(* PLC project Unnamed, Unnamed Unnamed 1 *)
(* stored: creationDateTime 2024-11-22T14:37:36, modificationDateTime 2024-11-29T13:18:13 *)

PROGRAM Blink
  VAR
    blink_led : BOOL;
    TON0 : TON;
    TOF0 : TOF;
    LED_ON0 : LED_ON;
    LED_OFF0 : LED_OFF;
    LED_ON1 : LED_ON;
    LED_OFF1 : LED_OFF;
  END_VAR
  VAR  (* added by the conversion: wires and edge detectors of the diagram *)
    R_TRIG1 : R_TRIG;
    F_TRIG2 : F_TRIG;
  END_VAR

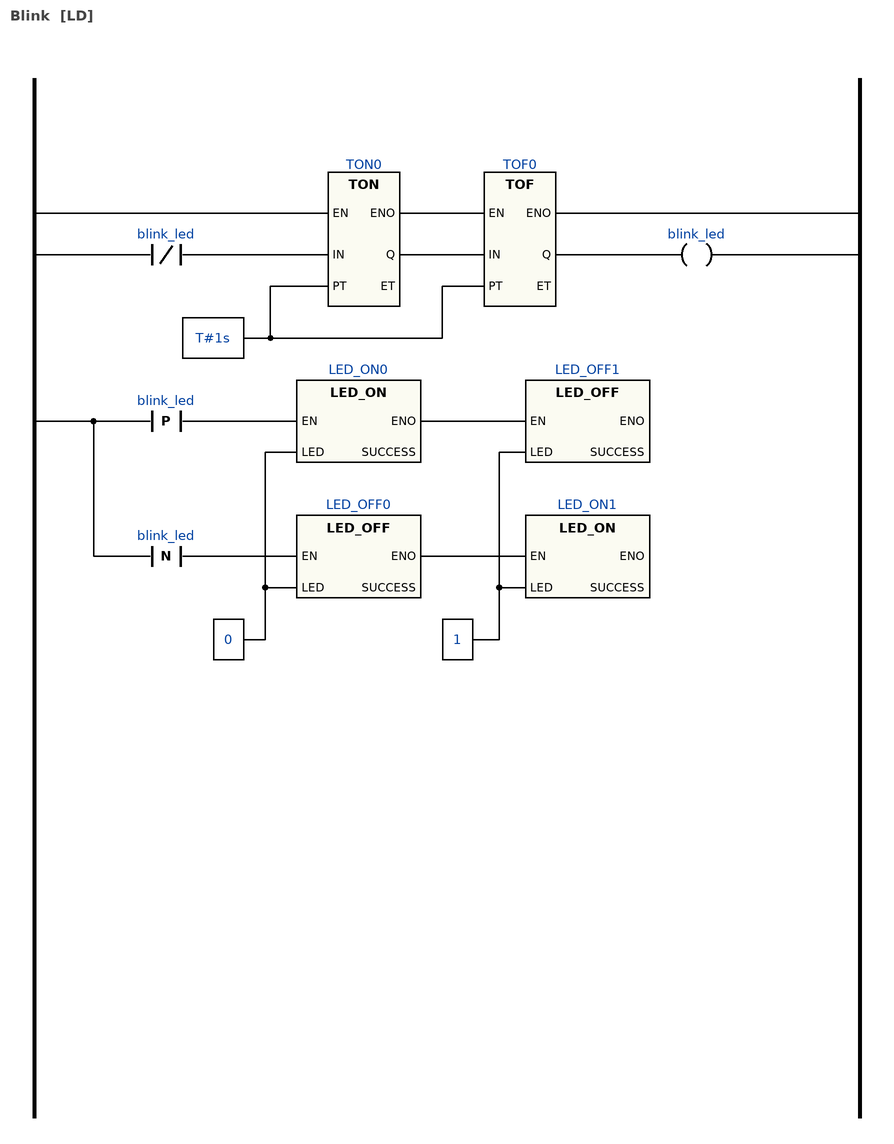
(* LD diagram, written out as Structured Text *)
TON0(IN := NOT blink_led, PT := T#1s);
TOF0(EN := TON0.ENO, IN := TON0.Q, PT := T#1s);
blink_led := TOF0.Q;
R_TRIG1(CLK := blink_led);
LED_ON0(EN := R_TRIG1.Q, LED := 0);
F_TRIG2(CLK := blink_led);
LED_OFF0(EN := F_TRIG2.Q, LED := 0);
LED_ON1(EN := LED_OFF0.ENO, LED := 1);
LED_OFF1(EN := LED_ON0.ENO, LED := 1);
END_PROGRAM

CONFIGURATION config
  RESOURCE resource1 ON PLC
    TASK task0(INTERVAL := T#50ms, PRIORITY := 0);
    PROGRAM instance0 WITH task0 : Blink;
  END_RESOURCE
END_CONFIGURATION
